SUBAPPLICATION Uebung_042 (* Scaling Function Block Testing *)
  (* Standard: 61499-2; Description: Copyright (c) 2023 Meisterschulen am Ostbahnhof This program and the accompanying materials are made available under the terms of the Eclipse Public License 2.0 which is available at https://www.eclipse.org/legal/epl-2.0/ SPDX-License-Identifier: EPL-2.0 *)
  (* Version 1.0, 2023-10-23, Franz Höpfinger, Meisterschulen am Ostbahnhof *)
  PACKAGE Uebungen;
  IMPORT logiBUS::io::DI::logiBUS_DI::Input_I1;
  IMPORT logiBUS::io::DI::logiBUS_DI_Events::BUTTON_SINGLE_CLICK;
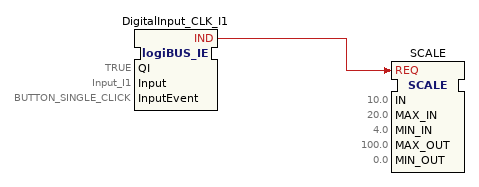
  FBS
    DigitalInput_CLK_I1 : logiBUS::io::DI::logiBUS_IE(QI := TRUE, Input := Input_I1, InputEvent := BUTTON_SINGLE_CLICK);
    SCALE : eclipse4diac::signalprocessing::SCALE(IN := 10.0, MAX_IN := 20.0, MIN_IN := 4.0, MAX_OUT := 100.0, MIN_OUT := 0.0);
  END_FBS
  EVENT_CONNECTIONS
    DigitalInput_CLK_I1.IND TO SCALE.REQ;
  END_CONNECTIONS
END_SUBAPPLICATION
